Universal Robots PolyScope program: testground.urp

Program testground (installation=mecspe_install directory=/home/ur/ursim-current/programs/mecspe2 createdIn=3.15.4.106291 lastSavedIn=3.15.4.106291 robotSerialNumber=2018359999)
Calibrated DH parameters: a=[0, -0.425, -0.39225, 0, 0, 0]; d=[0.089159, 0, 0, 0.10915, 0.09465, 0.0823]; alpha=[1.570796, 0, 0, 1.570796, -1.570796, 0]; deltaTheta=[0, 0, 0, 0, 0, 0]
Robot Program (runOnlyOnce=false)
  Script file /home/ur/ursim-current/programs/relPose.script
    | def relPose(FeaturePose,vect):
    | 
    |     # FeaturePose is the pose for the feature
    |     # vect = p[0.1, 0, 0, 0, 0, 0] makes us move 10cm in the X direction of the feature
    |     # credits: https://forum.universal-robots.com/t/move-tcp-relative-to-feature/15492
    | 
    |    PoseRelativeToFeature = pose_trans(pose_inv(FeaturePose), get_actual_tcp_pose())
    |    MoveTCPRelativeToFeature = pose_add(PoseRelativeToFeature, vect)
    |    return pose_trans(FeaturePose, MoveTCPRelativeToFeature)
    | 
    | end
  Script file /home/ur/ursim-current/programs/mecspe2/pose_to_position.script
    | def calc_pose_to_position(pose, feature, position):
    | 
    |    PoseRelativeToFeature = pose_trans(pose_inv(feature), pose)
    | 
    |    diff = pose_sub(position, PoseRelativeToFeature)
    |    vect = p[diff[0], diff[1], diff[2], 0, 0, 0]
    | 
    |    MoveTCPRelativeToFeature = pose_add(PoseRelativeToFeature, vect)
    |    return pose_trans(feature, MoveTCPRelativeToFeature)
    | 
    | end
  Script file /home/ur/ursim-current/programs/mecspe2/pose_trasf.script
    | def pose_trasf(pose, feature, vect):
    | 
    |    PoseRelativeToFeature = pose_trans(pose_inv(feature), pose)
    |    MoveTCPRelativeToFeature = pose_add(PoseRelativeToFeature, vect)
    |    return pose_trans(feature, MoveTCPRelativeToFeature)
    | 
    | end
  var_2 :=  (valueSource=Operator message=ask valueType=Integer)
  MoveJ speed 60 deg/s, acceleration 80 deg/s^2 (useActiveTCP=true)
    Waypoint Waypoint_1: TCP in base x=173.256 y=555.938 z=79.137 mm, rx=-2.9258 ry=-0.6294 rz=-0.5577 rad; joints [92.04, -115.02, -117.292, -28.081, 70.303, -23.911] deg; flange x=118.082 y=530.347 z=103.267 mm, rx=-2.9258 ry=-0.6294 rz=-0.5577 rad
    var_1 := pose_trasf(Waypoint_1,piano_moduli,p[0.1,0,0,0,0,0])
    Waypoint Waypoint (Variable): variable=var_1
    Waypoint Waypoint_2: TCP in base x=333.873 y=484.241 z=484.503 mm, rx=1.8885 ry=-0.5494 rz=2.238 rad; joints [77.966, -110.68, -90.438, -15.856, -12.891, -43.679] deg; flange x=301.604 y=506.502 z=432.116 mm, rx=1.8885 ry=-0.5494 rz=2.238 rad
    var_1 := pose_to_position(Waypoint_1,piano_moduli,p[0.1-0.07,-0.03,0.4,0,0,0])
    Waypoint Waypoint (Variable): variable=var_1
